TYPE ST_GS1_Decode_AI :
STRUCT
	sAI_Id		: STRING(5);
	bFixed		: BOOL;
	nLength		: UINT;
END_STRUCT
END_TYPE

(* stored: Version 1.1.0.1, ProductVersion 3.1.4024.15
   DUT ST_GS1_Decode_AI: Id {082f7c67-3f96-46c0-9461-6071fa4970b1} *)
